FUNCTION_BLOCK HaltTask EXTENDS TcoCore.TcoTask IMPLEMENTS IAxisIAI
VAR
    {attribute addProperty Name "<#Deceleration#>"}
    _deceleration : UINT;
END_VAR


IF Execute() THEN
    DriveRef.PlcToDrive.ControlSignal.STP := TRUE;

    DoneWhen(DriveRef.AxisStatus.NotMoving);
    ThrowWhen(DriveRef.AxisStatus.Error);
END_IF

PROPERTY DriveRef : REFERENCE TO AxisIAI
GET
VAR
    _drive : POINTER TO AxisIAI;
END_VAR
IF __QUERYPOINTER(THIS^._ParentObject, _drive) THEN
    DriveRef REF= _drive^;
END_IF
END_GET
END_PROPERTY

METHOD PUBLIC FB_init : BOOL
VAR_INPUT
    bInitRetains : BOOL; // if TRUE, the retain variables are initialized (warm start / cold start)
    bInCopyCode  : BOOL; // if TRUE, the instance afterwards gets moved into the copy code (online change)
    ParentObject : ITcoObject;
END_VAR
SUPER^.FB_init(bInitRetains := bInitRetains, bInCopyCode := bInCopyCode, ParentObject := ParentObject);
END_METHOD

METHOD INTERNAL InvokeWithParams : ITcoTaskStatus
VAR_INPUT
    inDeceleration : UINT;
END_VAR
_deceleration    := inDeceleration;
InvokeWithParams := THIS^.Invoke();
END_METHOD

(*~
    <docu>
        <summary>
            Executes when task reaches the ```Done``` state .
        </summary>
    </docu>
~*)
METHOD PROTECTED OnDone
Restore();
DriveRef.Restore();
END_METHOD

(*~
    <docu>
        <summary>
            Restores this instance to the Ready state. Can be called explicitly or from within one of the restore mechanisms.
            <para>
                See also <see cref="PlcDocu.TcoCore.TcoTask.AutoRestorable()"/>
            </para>
        </summary>
    </docu>
~*)
METHOD Restore : ITcoRestorable
SUPER^.Restore();
END_METHOD

END_FUNCTION_BLOCK

(* stored: Version 1.1.0.1, ProductVersion 3.1.4024.12
   POU HaltTask: Id {bb16a131-b32c-4030-a522-c95814497b94}, SpecialFunc None
   Property DriveRef: Id {c59ec605-f030-490f-b923-419033315d97}
   Get Get: Id {054177ef-c78a-48e0-adb3-b81e9bc991a3}
   Method FB_init: Id {12d8a9e1-892d-4869-9e34-0117ae4179d4}
   Method InvokeWithParams: Id {20c38d15-1ed1-48af-89be-20c9e33cad77}
   Method OnDone: Id {1f7c4a2c-2e9e-4437-94d4-bc2c693b4cbd}
   Method Restore: Id {9b2ea95e-7f3f-4504-980e-642478300964} *)
